FUNCTION_BLOCK Test_TStreamAdd_Read_UDINT_CheckAlignment EXTENDS T_UnitTestBase
VAR
    Stream  : T_Stream(StreamLength := 2);
    ArgType : E_ArgTypeId := E_ArgTypeId.Type_UDINT;
END_VAR

{attribute 'analysis' := '-33'} // inhibit unused variable warning
METHOD RunTest
Stream.Init(2);

Stream.Add_BYTE(123);// add a byte to test alignment checks...
Stream.Add_UDINT(12345678);

Stream.SetReadPosition(0);

Stream.Read_BYTE();

// check next value...	
AssertEquals_UDINT(Expected     := 12345678,
                             Actual       := Stream.Read_UDINT(),
                             Message := 'Stream.Read_UDINT()');

// check we are at the end of the stream..							
AssertEquals_UDINT(Expected     := Stream.StreamLength,
                             Actual       := Stream.ReadPosition,
                             Message := 'Stream.ReadPosition');

TestCompleted := TRUE;
END_METHOD

END_FUNCTION_BLOCK

(* stored: Version 1.1.0.1, ProductVersion 3.1.4024.12
   POU Test_TStreamAdd_Read_UDINT_CheckAlignment: Id {aa11c760-e2d4-43bf-9a04-772723f04080}, SpecialFunc None
   Method RunTest: Id {71474bb8-022e-43b2-9a11-6c6c4cd24373} *)
